// TIA Portal V19 export
FUNCTION_BLOCK "VSD Item Control"   // FB4, STL
{ S7_Optimized_Access := 'TRUE' }
// Flag uses in function
// M 4.0 - 1HZ onshot trigger bit (uses to count in seconds)
// 
// M 6.0 - set if new feedback alarm (used to activate alarm flash lamp)
// 
// 
// Data words uses in function
// 
// DB10, dw X - command word from SCADA
// Bit 0 = auto
// Bit 1 = Manuel deactivate
// Bit 2 = Manuel activate
// Bit 3 = spare
// Bit 4 = spare
// Bit 5 = spare
// Bit 6 = spare
// 
// DB11, dw X - info word to SCADA
// Bit 0  = activated
// Bit 1  = changing
// Bit 2  = faulty 
// Bit 3  = auto_man, Manual = 1 
// Bit 4  = man_on_off
// Bit 5  = Reset_FB
// Bit 6  = ManualSelected
// Bit 7  = Set_FB
// Bit 8  = Locate Active 
// Bit 9  = TrippedInd 
// Bit 10 = IsolatedInd 
// Bit 11 = VSD_Fault  
// Bit 12 = VSD_Alarm 
// Bit 13 = sv_3Activated 
// Bit 14 = fb_error - Alarm feedback error
// Bit 15 = sv_2Activated  
//  
// 
// DB13 byte x & byte x+1 - Timer work area
// Byte x   = spare     
// Byte x+1 = fb_timer    - Feedback timer item
// 
// DB 14, bit 0 - 7 & byte X+1 - Intern status & communication to monitor 
// functions 
// Bit 0  = spare
// Bit 1  = spare
// Bit 2  = spare
// Bit 3  = process_req - Process request from functions
// Bit 4  = process_mirror1 - Mirror process request
// Bit 5  = spare
// Bit 6  = spare
// Bit 7  = spare
// 
// Byte x+1 alarm_reset_timer alarm bit reset time 
// Bit 0-3  spare
// Bit 4-7  alarm reset timer for feedback error
// stored: AutoNumber false, MemoryReserve 100
   VAR_INPUT
      tripped : Bool;   // MPCB tripped
      iso_On : Bool;   // Local Isolator ON
      maxTime : Int;   // MAX FEED-BACK TIME
      rpm_Sp : Real;   // VSD RPM setpoint
      hwID : HW_ANY;   // IO Address on VSD
   END_VAR
   VAR_IN_OUT
      output : Bool;   // OUTPUT
      ItemInfo : "ItemInfo_UDT";
      ItemTimer : "ItemTimer_UDT";
      ItemStatus : "ItemStatus_UDT";
      ItemCommand : "ItemCommand_UDT";
   END_VAR
   VAR
      vsd { S7_SetPoint := 'True'} : SinaSpeed;
      ActualSpeed : Real;
   END_VAR
BEGIN

NETWORK
TITLE = ACTUATING
// CONTROL OUTPUT
      AN    #ItemInfo.auto_man;  // IF AUTO
      A     #ItemStatus.Auto;  // AND ProcessReq
      O(;
      A     #ItemInfo.auto_man;  // IF Manuel
      A     #ItemInfo.man_on_off;  // Manuel on/off
      );
      AN    #tripped;
      A     #iso_On;
      AN    #vsd.Error;
      AN    #vsd.Lockout;
      =     #output;  // Set/reset Output
//;


NETWORK
TITLE = CHANGE CONTROL
// CHANGE CONTROL
      A     #ItemStatus.Auto;  // IF ProcessReq
      AN    #ItemStatus.Process_Mirror;  // AND NOT PRMirror
      O(;  // OR
      AN    #ItemStatus.Auto;  // IF NOT ProcessReq
      A     #ItemStatus.Process_Mirror;  // AND PRMirror
      );
      JC    L1;  // Goto L1
      JU    NEX3;  //NEXT;        // ELSE Next
//;                      // ================================
L1:   L     0;  // Reset FeedbackTimer
      T     #ItemTimer.fb_timer;
//;
      A     #ItemStatus.Auto;
      =     #ItemStatus.Process_Mirror;  // PRMirror=ProcessReq
//;
NEX3: NOP   0;

NETWORK
TITLE = SCADA INFO & command
// Scada info and command
// 
// 
// ;=========================== Scada command ================================
//    OPN   "ItemCommand"               // SCADA COMMAND DB
      AN    #ItemCommand.Auto;
      AN    #ItemCommand.Locate;
      AN    #ItemCommand.Man_Act;
      AN    #ItemCommand.Man_DeAct;
      AN    #ItemCommand.Teach;
      AN    #ItemCommand.SpareBool;
      AN    #ItemCommand.SpareBool_1;
      AN    #ItemCommand.SpareBool_2;
      AN    #ItemCommand.SpareBool_3;
      AN    #ItemCommand.SpareBool_4;
      AN    #ItemCommand.SpareBool_5;
      AN    #ItemCommand.SpareBool_6;
      AN    #ItemCommand.SpareBool_7;
      AN    #ItemCommand.SV_2SelectionBit;
      AN    #ItemCommand.SV_3SelectionBit;
      AN    #ItemCommand.SpareBool_10;
      JC    INFO;  // if commamd bits = 0 then no commands

      A     #ItemCommand.Auto;
      R     #ItemInfo.auto_man;  // Auto/manual
      JC    clea;  // jump to clear command word

      A     #ItemCommand.Man_DeAct;
      S     #ItemInfo.auto_man;  // Auto/manual
      R     #ItemInfo.man_on_off;  // manual on/off
      JC    clea;  // jump to clear command word

      A     #ItemCommand.Man_Act;
      S     #ItemInfo.auto_man;  // Auto/manual
      S     #ItemInfo.man_on_off;  // manual on/off
      JC    clea;  // jump to clear command word

clea: SET;
      R     #ItemCommand.Auto;
      R     #ItemCommand.Locate;
      R     #ItemCommand.Man_Act;
      R     #ItemCommand.Man_DeAct;
      R     #ItemCommand.Teach;
      R     #ItemCommand.SpareBool;
      R     #ItemCommand.SpareBool_1;
      R     #ItemCommand.SpareBool_2;
      R     #ItemCommand.SpareBool_3;
      R     #ItemCommand.SpareBool_4;
      R     #ItemCommand.SpareBool_5;
      R     #ItemCommand.SpareBool_6;
      R     #ItemCommand.SpareBool_7;
      R     #ItemCommand.SV_2SelectionBit;
      R     #ItemCommand.SV_3SelectionBit;
      R     #ItemCommand.SpareBool_10;

//;=========================== Scada info ================================
INFO: A     #ItemInfo.fb_error;  // feedback error
      =     #ItemInfo.faulty;
      A     #ItemInfo.auto_man;
      =     #ItemInfo.ManualSelected;  //Show Manual selected on SCADA

// Set_FB off Actual Speed of motor
      L     #ActualSpeed;
      L     0;
      <>I;
      JCN   nrot;
      =     #ItemInfo.Set_FB;  //Show Set FB in "Item Info & Operation" popup
      R     #ItemInfo.Reset_FB;
      JU    rot;
nrot: =     #ItemInfo.Reset_FB;  //Show Reset FB in "Item Info & Operation" popup
      R     #ItemInfo.Set_FB;
rot:  A     #tripped;
      =     #ItemInfo.TrippedInd;
      AN    #iso_On;
      =     #ItemInfo.IsolatedInd;


      A     #output;  // IF Output
      AN    #ItemInfo.Set_FB;  // AND NOT SetFB
      JC    CHAN;  // Goto Changing
      A     #output;  // IF Output                       // AND SetFB
      A     #ItemInfo.Set_FB;
      JC    ACT;  // Goto Activated
      JU    DEAC;

//;                     // ================================
DEAC: R     #ItemInfo.activated;  // Update = deactivated
      R     #ItemInfo.changing;
      JU    NEX4;  //NEXT;
//;                     // ================================
CHAN: R     #ItemInfo.activated;  // Update = activated
      S     #ItemInfo.changing;
      JU    NEX4;  //NEXT;
//;                     // ================================
ACT:  S     #ItemInfo.activated;  // Update = activated
      R     #ItemInfo.changing;
      JU    NEX4;  //NEXT;
//;                     // ================================
NEX4: NOP   0;

NETWORK
TITLE = CONT.MONITORING
// FEEDBACK TEST
      AN    "1hz_oneshot_valve handle";  // IF NOT TimeSec
      JC    NEX5;  //NEXT;       // Goto Next
//;                     // ================================

// IF Type=SetFB
      A     #output;  // IF Output
      A     #ItemInfo.Set_FB;  // AND SetFB
      O;  //OK;         // Goto OK
      AN    #output;  // IF NOT Output
      AN    #ItemInfo.Set_FB;  // AND NOT SetFB
      JC    OK5;  //OK;         // Goto OK
      JU    CHAL;  // Else goto CheckAlarm

OK5:  L     0;
      T     #ItemTimer.fb_timer;  // Reset TimeCont.
// Reset Cont.Error
      JU    NEX5;  //NEXT;
//;                     // ================================
CHAL: L     #ItemTimer.fb_timer;  // Adjust TimeCont.
      INC   1;
      T     #ItemTimer.fb_timer;
      L     100;
      <=I;
      JC    CH1;
      L     100;
      T     #ItemTimer.fb_timer;
//;                     // ================================
CH1:  L     #ItemTimer.fb_timer;  // IF TimeCont. >=
      L     #maxTime;  // Max feedback time
      >=I;
      JC    ALRM;  // Goto Alarm
// Reset Cont.Error
      JU    NEX5;  //NEXT;
//;                     // ================================

ALRM: AN    #ItemInfo.fb_error;  // Set Cont.Error
      S     "Set_alarm_lamp_monitor";  // If new monitor alarm set alarm flash lamp
      SET;
      S     #ItemInfo.fb_error;  // Set Cont.Error
//
      L     #ItemStatus.AlarmResetTimer;
      L     16#0050;  // Wait 5 seconds to reset alarm bits
      OW;  // Larst 4 bits time reset monitor/process alarm
      T     #ItemStatus.AlarmResetTimer;
//;                     // ================================
NEX5: NOP   0;

NETWORK
TITLE = Reset alarm bits
// Reset alarm bit after 5 seconds
      AN    "1hz_oneshot_valve handle";  // IF NOT TimeSec
      JC    nex6;  // Goto Next
//;                     // ================================
      L     #ItemStatus.AlarmResetTimer;

      L     16#00F0;  // larst 4 bit in byte = counter
      AW;
      L     0;
      ==I;  // alarm high in min 5 seconds
      R     #ItemInfo.fb_error;  // Reset Cont.Error
      JC    nex6;
      L     #ItemStatus.AlarmResetTimer;
      L     16#0010;  // Count 1 second down, in larst 4 bit time reset F.B. alarm
      -I;
      T     #ItemStatus.AlarmResetTimer;
nex6: NOP   0;

NETWORK
TITLE = vsd block
      CALL  #vsd
      ( EnableAxis  := #output,
        AckError    := ,
        SpeedSp     := #rpm_Sp,
        RefSpeed    := 1460.0,
        ConfigAxis  := ,
        HWIDSTW     := #hwID,
        HWIDZSW     := #hwID,
        AxisEnabled := #output,
        Lockout     := ,
        ActVelocity := #ActualSpeed,
        Error       := #ItemInfo.VSD_Fault,
        Status      := ,
        DiagId      := 
      );


END_FUNCTION_BLOCK
